FUNCTION_BLOCK TestWrapper
VAR
	core_logger : TcLogCore(BufferSize:=50 * 50 * (Tc2_System.MAX_STRING_LENGTH + Constants.FifoOverhead));
	core_logger_first_cycle : TcLogCore(BufferSize:=50 * 50 * (Tc2_System.MAX_STRING_LENGTH + Constants.FifoOverhead));
	core_logger_first_cycle_valid_timestamp_only : TcLogCore(BufferSize:=50 * 50 * (Tc2_System.MAX_STRING_LENGTH + Constants.FifoOverhead));
	logger_first_cycle : TcLog;
	logger_first_cycle_valid_timestamp_only : TcLog;
	logger : TcLog;
	flush_cache : BOOL;
	ads_adapter : AdsLogTargetAdapter;
 
	// Test drivers
	date_time : DateTime;
	set_local_system_time : NT_SetLocalTime;
	cycles : INT;
	_i : INT;
	persistence_time_stays_within_bounds : F_Trig;
	is_first_cycle: BOOL := TRUE;
	
	// Exchanged variables with .NET tests
	FilePath : STRING;
	FileName : STRING;
	Delimiter : STRING(1);
	NewLocalSystemTimeToBeSet : STRING;
	TriggerNewLocalSystemTime : BOOL;
	LocalTimeAsString : STRING;
	
	Persist_simple_error_message_run : BOOL;
	Persist_simple_error_message_data : STRING;
	
	Persist_long_error_message_run : BOOL;
	Persist_long_error_message_data : T_MaxString;
	
	Linebreak_is_included_when_log_message_has_maximum_length_run : BOOL;
	Linebreak_is_included_when_log_message_has_maximum_length_data : T_MaxString;
	
	Do_not_persist_logs_below_log_level_run : BOOL;
	
	Log_message_contains_instance_path_run : BOOL;
	
	Log_message_uses_correct_delimiter_run : BOOL;
	Log_message_uses_correct_delimiter_data : STRING;
	
	Log_message_contains_custom_formatted_timestamp_run : BOOL;
	
	Delete_logs_if_expired_run : BOOL;
	
	New_logfile_is_created_if_rolling_interval_rolls_run : BOOL;
	
	Same_log_file_is_used_until_rolling_interval_rolls : BOOL;
	
	Log_in_consecutive_cycles : BOOL;
	Number_of_log_cycles : DINT;
	
	Log_multiple_logs_in_one_cycle : BOOL;
	Number_of_logs_per_cycle : DINT;
	
	Log_multiple_logs_in_multiple_cycles : BOOL;
	Number_of_cycles : DINT;
	CycleCount : DINT := 1;
	
	Persistance_time_stays_within_bounds : BOOL;
	Duration_in_cylces : DINT := 1;
END_VAR

// ****** U N I T   T E S T S ******

// Set up TcLog
core_logger
	.IncludeInstancePath()
	.MinimumLevel(LogLevel.Debug)
	.SetDelimiter(Delimiter)
	.SetRollingInterval(RollingIntervals.Hourly)
	.DeleteLogFilesAfterDays(1)
	.TimestampFormat('_YYMMDD-hh-mm-ss_')
	.WriteToAds()
	.WriteToFile('C:\Log Files', 'tclog_test.log')
	.WriteToAdapter(ads_adapter)
	.RunLogger();
//logger.SetLogger(core_logger);

IF flush_cache THEN
	core_logger.FlushCache();
END_IF
  
// Test drivers
date_time.CyclicCall();
LocalTimeAsString := date_time.AsLocalSystemTimeString;

set_local_system_time(
	NetId   := '',
	TimeStr := STRING_TO_SYSTEMTIME(NewLocalSystemTimeToBeSet),
	Start   := TriggerNewLocalSystemTime,
	TmOut := T#2S
);

// Execute tests
IF Persist_simple_error_message_run THEN
	Persist_simple_error_message_run := FALSE;
	logger.Error(Persist_simple_error_message_data);
END_IF

IF Persist_long_error_message_run THEN
	Persist_long_error_message_run := FALSE;
	logger.ToCustomFormat(Persist_long_error_message_data);
END_IF

IF Linebreak_is_included_when_log_message_has_maximum_length_run THEN
	Linebreak_is_included_when_log_message_has_maximum_length_run := FALSE;
	logger
		.ToCustomFormat(Linebreak_is_included_when_log_message_has_maximum_length_data);
	logger.ToCustomFormat(Linebreak_is_included_when_log_message_has_maximum_length_data);
END_IF

IF Do_not_persist_logs_below_log_level_run THEN
	Do_not_persist_logs_below_log_level_run := FALSE;
	logger.Information('Nothing');
END_IF

IF Log_message_contains_instance_path_run THEN
	Log_message_contains_instance_path_run := FALSE;
	logger.Error('Nothing');
END_IF

IF Log_message_uses_correct_delimiter_run THEN
	Log_message_uses_correct_delimiter_run := FALSE;
	logger.Error(Log_message_uses_correct_delimiter_data);
END_IF

IF Log_message_contains_custom_formatted_timestamp_run THEN
	Log_message_contains_custom_formatted_timestamp_run := FALSE;
	logger.Error('Test message');
END_IF

IF Delete_logs_if_expired_run THEN
	Delete_logs_if_expired_run := FALSE;
	logger.Error('Test message');
END_IF

IF New_logfile_is_created_if_rolling_interval_rolls_run THEN
	New_logfile_is_created_if_rolling_interval_rolls_run := FALSE;
	logger.Error('Test message');
END_IF

IF Same_log_file_is_used_until_rolling_interval_rolls THEN
	Same_log_file_is_used_until_rolling_interval_rolls := FALSE;
	logger.Error('Test message');
END_IF

IF Log_in_consecutive_cycles THEN
	logger.Error(Tc2_Standard.CONCAT('Logging cycle ', INT_TO_STRING(cycles)));
	cycles := cycles + 1;
	IF cycles >= Number_of_log_cycles THEN
		cycles := 0;
		Log_in_consecutive_cycles := FALSE;
	END_IF
END_IF

IF Log_multiple_logs_in_one_cycle THEN
	FOR _i:= 1 TO DINT_TO_INT(Number_of_logs_per_cycle) DO
		logger.
			Error(Tc2_Standard.CONCAT('Logging multiple times per cycle. Current step: ', INT_TO_STRING(_i))); 
	END_FOR
	Log_multiple_logs_in_one_cycle := FALSE;
END_IF

IF Log_multiple_logs_in_multiple_cycles THEN
	IF CycleCount <= Number_of_cycles THEN  
		FOR _i:= 1 TO DINT_TO_INT(Number_of_logs_per_cycle) DO
			logger
				.AppendString('Logging multiple times per cycle. Cycle: ')
				.AppendString(DINT_TO_STRING(CycleCount))
				.AppendString(' / Step: ')
				.AppendString(INT_TO_STRING(_i))
				.Error('');
		END_FOR
		CycleCount := CycleCount + 1;
	ELSE
		CycleCount := 1;
		Log_multiple_logs_in_multiple_cycles := FALSE;
	END_IF
END_IF 

persistence_time_stays_within_bounds(CLK := (Persistance_time_stays_within_bounds AND core_logger.Busy));
IF persistence_time_stays_within_bounds.Q THEN
	CycleCount := 1;
	Persistance_time_stays_within_bounds := FALSE;
END_IF

IF Persistance_time_stays_within_bounds THEN
	Duration_in_cylces := Duration_in_cylces + 1;
	IF CycleCount <= Number_of_cycles THEN  
		FOR _i:= 1 TO DINT_TO_INT(Number_of_logs_per_cycle) DO
			logger
				.AppendString('Logging multiple times per cycle. Cycle: ')
				.AppendString(DINT_TO_STRING(CycleCount))
				.AppendString(' / Step: ')
				.AppendString(INT_TO_STRING(_i))
				.Error('');
		END_FOR
		CycleCount := CycleCount + 1;
	END_IF
END_IF

// Check first cpu cycle
core_logger_first_cycle
	.IncludeInstancePath()
	.MinimumLevel(LogLevel.Warning)
	.SetDelimiter(Delimiter)
	.SetRollingInterval(RollingIntervals.Hourly)
	.DeleteLogFilesAfterDays(1)
	.TimestampFormat('_YYYYMMDD-hh-mm-ss_')
	.WriteToAds()
	.WriteToFile('C:\UnitTestFirstCycle\', 'firstCycle.txt')
	.RunLogger();
logger_first_cycle.SetLogger(core_logger_first_cycle);

core_logger_first_cycle_valid_timestamp_only
	.IncludeInstancePath()
	.MinimumLevel(LogLevel.Warning)
	.SetDelimiter(Delimiter)
	.SetRollingInterval(RollingIntervals.Hourly)
	.DeleteLogFilesAfterDays(1)
	.TimestampFormat('_YYYYMMDD-hh-mm-ss_')
	.WriteToAds()
	.WriteToFile('C:\UnitTestFirstCycle\', 'firstCycleValidTimestampOnly.txt')
	.ValidTimestampsOnly()
	.RunLogger();
logger_first_cycle_valid_timestamp_only.SetLogger(core_logger_first_cycle_valid_timestamp_only);

IF is_first_cycle THEN
	logger_first_cycle.Error('Log in first cycle');
	logger_first_cycle_valid_timestamp_only.Error('Log in first cycle with valid timestamps only');
	is_first_cycle := FALSE;
END_IF

END_FUNCTION_BLOCK

(* stored: Version 1.1.0.1, ProductVersion 3.1.4026.17
   POU TestWrapper: Id {2083d311-1ce0-4edb-9acc-97906d1cd251}, SpecialFunc None *)
